{attribute addProperty BoxType "AMP8000-0030-0103-0103"}
{attribute addProperty Id "FSOEAT %I*FSOE_712CBB49567"}
{attribute addProperty CRC "4112596503"}
{attribute addProperty SizeInBites "56"}
{attribute addProperty SizeInBytes "7"}
TYPE FSoE_Slave_Connection_1_Slave_Message_F5213E17 :
STRUCT
	{attribute addProperty Name "FSOE"}
	FSOE AT %I* : FSOE_712CBB49;
END_STRUCT
END_TYPE

(* stored: Version 1.2.0.0, ProductVersion 3.1.4024.9
   DUT FSoE_Slave_Connection_1_Slave_Message_F5213E17: Id {af9743af-c780-4910-be63-e88b313f1c01} *)
